// TIA Portal V20 export
TYPE "RollBed"
   STRUCT
      HMI : "H_HMI";
      G120 { S7_SetPoint := 'True'} : "H_Roller2W2S-G120PN";
      Config { S7_SetPoint := 'True'} : "RollerConvConfig";
      InPut : "InPut";
      OutPut : "OutPut";
   END_STRUCT;
END_TYPE
